Yaskawa INFORM job: WILL.JBI

/JOB
//NAME WILL
//POS
///NPOS 5,0,0,0
///TOOL 0
///PULSE
C000=46767,31765,-45867,9545,9957,7922
C001=46767,31765,-16683,9545,9957,7922
C002=46767,31765,-16347,9545,9957,10806
C003=34479,31765,-16347,7025,9957,10806
C004=34479,16837,-16347,7025,9957,10806
//INST
///DATE 2014/09/16 21:22
///ATTR 0,0,0,0,0,0,0,0,0,0,0,0,0,1,0,0
///FRAME BASE
NOP
*L
MOVJ C000 VJ=100.00 CONT
MOVJ C001 VJ=100.00 CONT
MOVJ C002 VJ=100.00 CONT
MOVJ C003 VJ=100.00 CONT
MOVJ C004 VJ=100.00 CONT
JUMP *L
END
